% RSLogix 500 project PROJECT8.RSS, saved by version 8.30.00.16 %
PROJECT "PROJECT8"    % processor: Bul.1763 MicroLogix 1100 Series B %

PROGRAM FILES
  LAD 2 "MAIN"  5 rungs
  LAD 3 "I/O"  2 rungs
  LAD 4 "RANGES"  4 rungs
  LAD 5 "PID"  6 rungs

DATA FILES
  O0 OUTPUT  6 elements
  I1 INPUT  12 elements
  S2 STATUS  66 elements
  B3 BINARY  1 elements
  T4 TIMER  1 elements
  C5 COUNTER  1 elements
  R6 CONTROL  1 elements
  N7 INTEGER  4 elements
  F8 FLOAT  12 elements

LADDER 2 "MAIN"
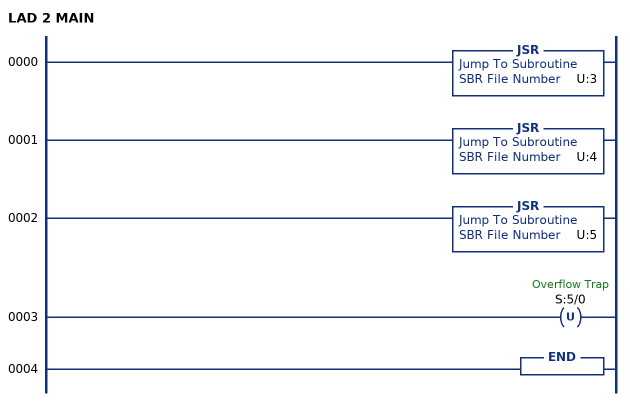
% Rung: 0 %
SOR JSR U:3 EOR
% Rung: 1 %
SOR JSR U:4 EOR
% Rung: 2 %
SOR JSR U:5 EOR
% Rung: 3 %
SOR OTU S:5/0 EOR
%   S:5/0  "Overflow Trap" %
% Rung: 4 %
SOR END EOR

LADDER 3 "I/O"
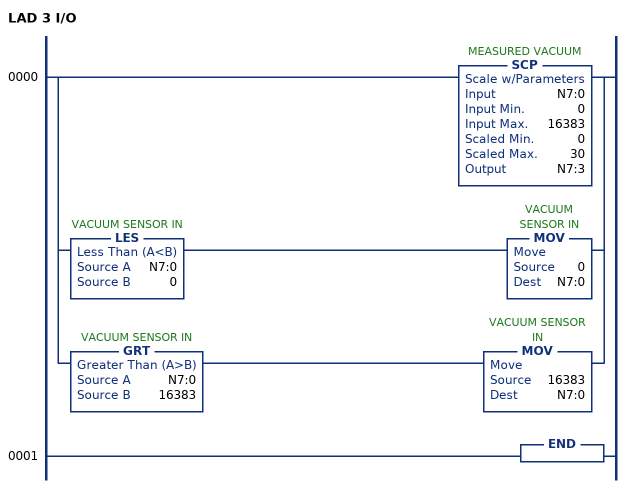
% Rung: 0 %
SOR BST SCP N7:0 0 16383 0 30 N7:3 NXB LES N7:0 0 MOV 0 N7:0 NXB GRT N7:0 16383 MOV 16383 N7:0 BND EOR
%   N7:0  "VACUUM SENSOR IN" %
%   N7:3  "MEASURED VACUUM" %
% Rung: 1 %
SOR END EOR

LADDER 4 "RANGES"
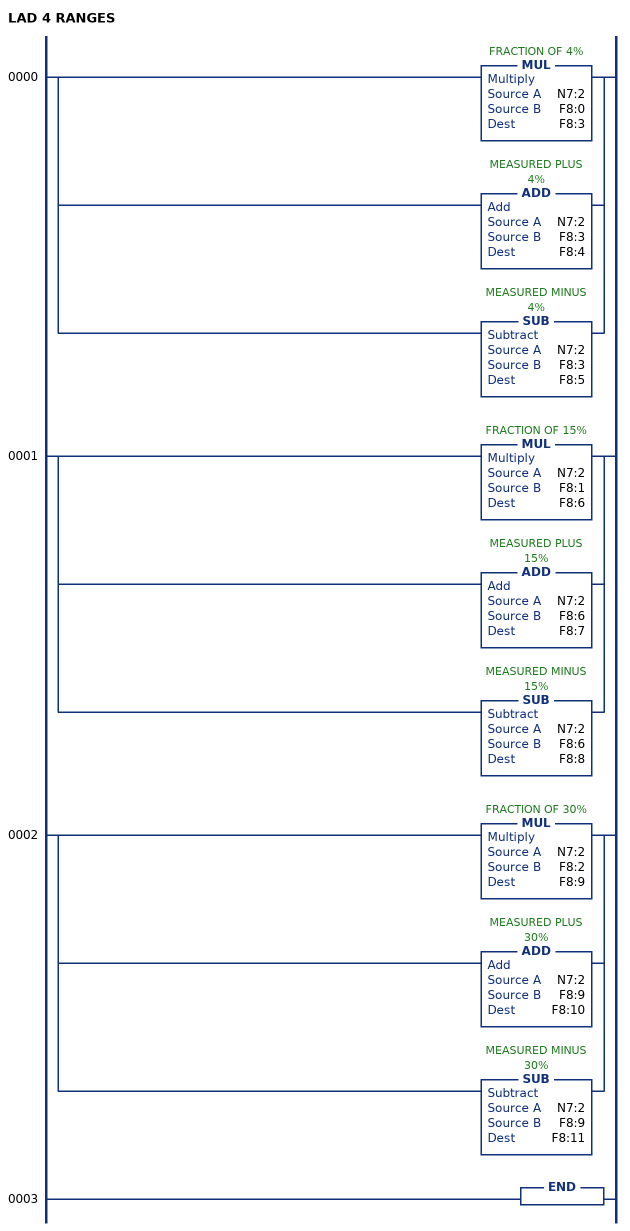
% Rung: 0 %
SOR BST MUL N7:2 F8:0 F8:3 NXB ADD N7:2 F8:3 F8:4 NXB SUB N7:2 F8:3 F8:5 BND EOR
%   N7:2  "VACUUM SETPOINT" %
%   F8:0  "RANGE 1" %
%   F8:3  "FRACTION OF 4%" %
%   F8:4  "MEASURED PLUS 4%" %
%   F8:5  "MEASURED MINUS 4%" %
% Rung: 1 %
SOR BST MUL N7:2 F8:1 F8:6 NXB ADD N7:2 F8:6 F8:7 NXB SUB N7:2 F8:6 F8:8 BND EOR
%   N7:2  "VACUUM SETPOINT" %
%   F8:1  "RANGE 2" %
%   F8:6  "FRACTION OF 15%" %
%   F8:7  "MEASURED PLUS 15%" %
%   F8:8  "MEASURED MINUS 15%" %
% Rung: 2 %
SOR BST MUL N7:2 F8:2 F8:9 NXB ADD N7:2 F8:9 F8:10 NXB SUB N7:2 F8:9 F8:11 BND EOR
%   N7:2  "VACUUM SETPOINT" %
%   F8:2  "RANGE 3" %
%   F8:9  "FRACTION OF 30%" %
%   F8:10  "MEASURED PLUS 30%" %
%   F8:11  "MEASURED MINUS 30%" %
% Rung: 3 %
SOR END EOR

LADDER 5 "PID"
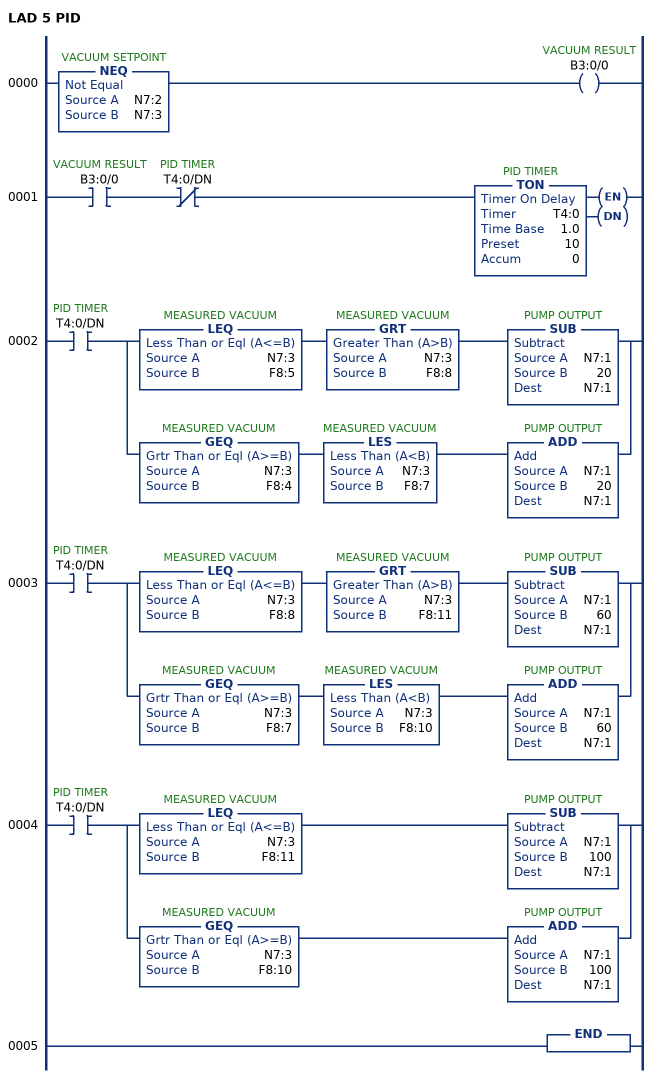
% Rung: 0 %
SOR NEQ N7:2 N7:3 OTE B3:0/0 EOR
%   N7:2  "VACUUM SETPOINT" %
%   N7:3  "MEASURED VACUUM" %
%   B3:0/0  "VACUUM RESULT" %
% Rung: 1 %
SOR XIC B3:0/0 XIO T4:0/DN TON T4:0 1.0 10 0 EOR
%   B3:0/0  "VACUUM RESULT" %
%   T4:0  "PID TIMER" %
% Rung: 2 %
SOR XIC T4:0/DN BST LEQ N7:3 F8:5 GRT N7:3 F8:8 SUB N7:1 20 N7:1 NXB GEQ N7:3 F8:4 LES N7:3 F8:7 ADD N7:1 20 N7:1 BND EOR
%   T4:0  "PID TIMER" %
%   N7:3  "MEASURED VACUUM" %
%   F8:5  "MEASURED MINUS 4%" %
%   F8:8  "MEASURED MINUS 15%" %
%   N7:1  "PUMP OUTPUT" %
%   F8:4  "MEASURED PLUS 4%" %
%   F8:7  "MEASURED PLUS 15%" %
% Rung: 3 %
SOR XIC T4:0/DN BST LEQ N7:3 F8:8 GRT N7:3 F8:11 SUB N7:1 60 N7:1 NXB GEQ N7:3 F8:7 LES N7:3 F8:10 ADD N7:1 60 N7:1 BND EOR
%   T4:0  "PID TIMER" %
%   N7:3  "MEASURED VACUUM" %
%   F8:8  "MEASURED MINUS 15%" %
%   F8:11  "MEASURED MINUS 30%" %
%   N7:1  "PUMP OUTPUT" %
%   F8:7  "MEASURED PLUS 15%" %
%   F8:10  "MEASURED PLUS 30%" %
% Rung: 4 %
SOR XIC T4:0/DN BST LEQ N7:3 F8:11 SUB N7:1 100 N7:1 NXB GEQ N7:3 F8:10 ADD N7:1 100 N7:1 BND EOR
%   T4:0  "PID TIMER" %
%   N7:3  "MEASURED VACUUM" %
%   F8:11  "MEASURED MINUS 30%" %
%   N7:1  "PUMP OUTPUT" %
%   F8:10  "MEASURED PLUS 30%" %
% Rung: 5 %
SOR END EOR

DATA TABLE (non-zero values as saved)
DATA T4
% .PRE .ACC %
% T4:0 % 10 0
DATA N7
% N7:0 % 0 0 15 0
DATA F8
% F8:0 % 0.04 0.15 0.3 0 0
